Staubli VAL3: sendInfo2Camera.pgx

program sendInfo2Camera()
  local num l_ns
  local string l_sData
begin
  l_sData=""
  skToCamera="start"
  l_ns=clock()
  do
    l_sData=skToCamera
    if (clock()-l_ns>1)
      call setAlarm(0)
    endIf
    delay(0)
  until (true)

end
